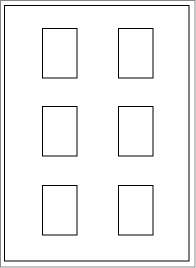
VISUALIZATION Carrinho  // 196x268
    RoundedRectangle (4,5 185x256)
    RoundedRectangle (35,36 50x35), angle 90, colour variable: GVL_P.corPosReator1[4].color
        OnMouseUp: execute { gvl.actReat:= 4; }
        OnMouseUp: OpenDialog Dialog=ConfigPosicao_Reator, Parameters={bReator: , iOFnumber: , iSrlNumber: }, OpenModal=True, OpenCentered=True
    RoundedRectangle (111,36 50x35), angle 90, colour variable: GVL_P.corPosReator1[1].color
        OnMouseUp: OpenDialog Dialog=ConfigPosicao_Reator, Parameters={bReator: , iOFnumber: , iSrlNumber: }, OpenModal=True, OpenCentered=True
        OnMouseUp: execute { gvl.actReat:= 1; posCarrinho(); }
    RoundedRectangle (111,114 50x35), angle 90, colour variable: GVL_P.corPosReator1[2].color
        OnMouseUp: execute { gvl.actReat:= 2; }
        OnMouseUp: OpenDialog Dialog=ConfigPosicao_Reator, Parameters={bReator: , iOFnumber: , iSrlNumber: }, OpenModal=True, OpenCentered=True
    RoundedRectangle (35,114 50x35), angle 90, colour variable: GVL_P.corPosReator1[5].color
        OnMouseUp: execute { gvl.actReat:= 5; }
        OnMouseUp: OpenDialog Dialog=ConfigPosicao_Reator, Parameters={bReator: , iOFnumber: , iSrlNumber: }, OpenModal=True, OpenCentered=True
    RoundedRectangle (111,193 50x35), angle 90, colour variable: GVL_P.corPosReator1[3].color
        OnMouseUp: execute { gvl.actReat:= 3; }
        OnMouseUp: OpenDialog Dialog=ConfigPosicao_Reator, Parameters={bReator: , iOFnumber: , iSrlNumber: }, OpenModal=True, OpenCentered=True
    RoundedRectangle (35,193 50x35), angle 90, colour variable: GVL_P.corPosReator1[6].color
        OnMouseUp: execute { gvl.actReat:= 6; }
        OnMouseUp: OpenDialog Dialog=ConfigPosicao_Reator, Parameters={bReator: , iOFnumber: , iSrlNumber: }, OpenModal=True, OpenCentered=True
END_VISUALIZATION

(* stored: Version 1.1.0.1, ProductVersion 3.1.4024.12
   Visu Carrinho: Id {42fd87d2-547f-450f-9e10-3c715ea95661} *)
